Fanuc KAREL source: kb00032.KL

-- PROVISIONAL review KL for V1013-1; original PC SHA256 7dd639b88493be010e03729c18c5e6a3cd61c901ae63f0f1ae04c288b99e4284
-- Incomplete behavior may be omitted. Consult companion uncertainty JSON. Do not deploy.
PROGRAM KB00032
%NOLOCKGROUP
BEGIN
  -- UNRESOLVED_PC offsets 5-14; opcodes 3F,75
  -- UNRESOLVED_PC offsets 19-28; opcodes 3F,75
  -- UNRESOLVED_PC offsets 33-40; opcodes 9D,23
  -- UNRESOLVED_PC offsets 45-71; opcodes 27,22,2A,22,2A,22,31
  -- UNRESOLVED_PC offsets 76-80; opcodes 7F
END KB00032
